SUBAPPLICATION Uebung_003c_AX (* DigitalInput_I1-2-3-4 auf AUX *)
  (* Standard: 61499-2; Description: Copyright (c) 2026 Meisterschulen am Ostbahnhof This program and the accompanying materials are made available under the terms of the Eclipse Public License 2.0 which is available at https://www.eclipse.org/legal/epl-2.0/ SPDX-License-Identifier: EPL-2.0 *)
  (* Version 1.0, 2026-01-13, Moritz Ortmeier, Meisterschulen am Ostbahnhof *)
  PACKAGE Uebungen;
  IMPORT logiBUS::io::DI::logiBUS_DI::Input_I1;
  IMPORT logiBUS::io::DI::logiBUS_DI::Input_I2;
  IMPORT logiBUS::io::DI::logiBUS_DI::Input_I3;
  IMPORT logiBUS::io::DI::logiBUS_DI::Input_I4;
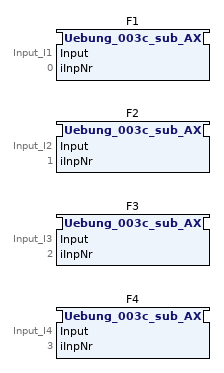
  SUBAPPS
    F1 : Uebungen::Uebung_003c_sub_AX(Input := Input_I1, iInpNr := 0);
    F2 : Uebungen::Uebung_003c_sub_AX(Input := Input_I2, iInpNr := 1);
    F3 : Uebungen::Uebung_003c_sub_AX(Input := Input_I3, iInpNr := 2);
    F4 : Uebungen::Uebung_003c_sub_AX(Input := Input_I4, iInpNr := 3);
  END_SUBAPPS
END_SUBAPPLICATION
